Yaskawa INFORM job: R2_W27-A3(90,0)_MP_OK.JBI

/JOB
//NAME R2_W27-A3(90,0)_MP_OK
///FOLDERNAME MP_TEST
//POS
///NPOS 44,44,0,2,0,0
///TOOL 0
///POSTYPE PULSE
///PULSE
C00000=101600,-116692,-81613,16390,61564,19311
C00001=164215,-55536,-44539,-18349,62898,27662
C00002=160924,-13115,576,-12085,68568,20289
C00003=160935,-12305,2800,-12163,67637,20390
C00004=160940,-12317,2798,-12164,67633,20392
C00005=160946,-12330,2788,-12165,67634,20394
C00006=160940,-12317,2798,-12164,67633,20392
C00007=160931,-12288,2814,-12162,67637,20389
C00008=160930,-12287,2823,-12162,67632,20389
C00009=160931,-12288,2814,-12162,67637,20389
C00010=160981,-12434,2698,-978,54579,-1424
C00011=160979,-12429,2730,-978,54561,-1425
C00012=160976,-12421,2736,-977,54562,-1426
C00013=160979,-12429,2730,-978,54561,-1425
C00014=160981,-12434,2698,-978,54579,-1424
C00015=160997,-12478,2668,-985,54575,-1417
C00016=160994,-12473,2666,-984,54579,-1419
C00017=160987,-12460,2661,-981,54588,-1422
C00018=145436,-5822,-19148,1406,76142,21143
C00019=161005,-17259,-14065,-3869,52708,76882
C00020=161000,-11415,3879,-4366,44687,77223
C00021=161004,-11424,3871,-4369,44687,77225
C00022=165127,-14952,4261,-15285,39692,81657
C00023=161056,-12333,1868,-4344,45453,77213
C00024=160458,-11230,5111,-4075,43997,76999
C00025=163098,-8602,9142,-13757,39586,80598
C00026=161003,-11423,3872,-4369,44687,77225
C00027=160999,-11413,3880,-4366,44687,77223
C00028=161005,-17410,-14659,-3854,52995,76871
C00029=116418,-11777,-44439,19300,59296,60154
C00030=170009,-32177,-45595,-27188,83944,54223
C00031=188971,-7216,-15050,-32227,103013,52664
C00032=187803,-7888,-16310,-32403,102934,52210
C00033=188364,-6082,-14100,-32286,102781,52484
C00034=188636,-9365,-17003,-32274,102969,52540
C00035=189413,-7325,-10428,-33924,100512,54745
C00036=189914,-7682,-12670,-35106,101599,55206
C00037=190540,-7572,-11965,-36074,101422,56128
C00038=193143,-7278,-8936,-40285,100522,60148
C00039=196044,-7471,-5630,-45187,99267,64707
C00040=192289,-11545,-19761,-34441,104887,54555
C00041=160924,-13115,576,-12085,68568,20289
C00042=164215,-55536,-44539,-18349,62898,27662
C00043=101600,-116692,-81613,16390,61564,19311
BC00000=282797,179500,1075171
BC00001=315243,149725,1075174
BC00002=326313,139566,1075175
BC00003=327306,134779,1064198
BC00004=327703,132864,1055897
BC00005=327690,132857,1047832
BC00006=327703,132864,1055897
BC00007=317158,132350,1053533
BC00008=317644,130094,1053548
BC00009=317158,132350,1053533
BC00010=354979,141253,1041870
BC00011=356652,133484,1041925
BC00012=354313,133016,1041973
BC00013=356652,133484,1041925
BC00014=354979,141253,1041870
BC00015=363025,141681,1030105
BC00016=364240,143651,1037263
BC00017=367279,148578,1055156
BC00018=320233,175848,913334
BC00019=353844,149726,1075175
BC00020=353886,149731,1052313
BC00021=353827,147577,1026510
BC00022=353804,146715,1016186
BC00023=353804,146715,1016188
BC00024=353804,146715,1016188
BC00025=353804,146715,1016186
BC00026=353799,139703,1029577
BC00027=353858,141857,1055381
BC00028=353816,141852,1075175
BC00029=253941,214275,713494
BC00030=305300,128666,812515
BC00031=329706,95698,858127
BC00032=329696,96061,851804
BC00033=329696,96061,851804
BC00034=329696,96061,851804
BC00035=329682,96606,842319
BC00036=329681,96639,841736
BC00037=329663,97291,830381
BC00038=329660,97348,828220
BC00039=329656,97223,825887
BC00040=329682,96606,842319
BC00041=326313,139566,1075175
BC00042=315243,149725,1075174
BC00043=282797,179500,1075171
///POSTYPE BASE
///RECTAN
///RCONF 0,0,0,0,1,0,0,0,0,0,0,0,0,0,0,0,0,0,0,0,0,0,0,0
P00006=2.006,1.622,-0.565,0.0000,0.0000,0.0000
///RCONF 0,0,0,0,0,0,0,0,0,0,0,0,0,0,0,0,0,0,0,0,0,0,0,0
P00014=4.542,-3.738,3.339,0.0000,0.0000,0.0000
//INST
///DATE 2023/11/16 10:45
///ATTR SC,RW
///GROUP1 RB1,BS1
NOP
'r2_W27-A3(90,0)
'
'Path S839
SFTOF
MOVJ C00000 BC00000 VJ=20.00
MOVJ C00001 BC00001 VJ=20.00
MOVL C00002 BC00002 V=100.0
MOVL C00003 BC00003 V=100.0
MOVL C00004 BC00004 V=60.0
REFP 3 C00005 BC00005
CALL JOB:SEARCH-R1
SET P014 P006
SFTON P014
MOVL C00006 BC00006 V=60.0
MOVL C00007 BC00007 V=60.0
REFP 3 C00008 BC00008
CALL JOB:SEARCH-R1
SET P014 P006
SFTON P014
MOVL C00009 BC00009 V=60.0
MOVL C00010 BC00010 V=100.0
MOVL C00011 BC00011 V=60.0
REFP 3 C00012 BC00012
CALL JOB:SEARCH-R1
SET P014 P006
SFTON P014
MOVL C00013 BC00013 V=60.0
MOVL C00014 BC00014 V=100.0
MOVL C00015 BC00015 V=100.0
MOVL C00016 BC00016 V=100.0
MOVL C00017 BC00017 V=100.0
'Path VIA886
SFTOF
MOVJ C00018 BC00018 VJ=20.00
'Path W840
SFTOF
SFTON P014
'ZA DUZA SZCZELINA
'ZA DUZA SZCZELINA
'ZA DUZA SZCZELINA
MOVJ C00019 BC00019 VJ=20.00
MOVJ C00020 BC00020 VJ=20.00
MOVL C00021 BC00021 V=100.0
MOVL C00022 BC00022 V=100.0 PL=0
REFP 1 C00023 BC00023
REFP 2 C00024 BC00024
MACRO1 MJ#(0) ARGF7
COMM ARCON
MOVL C00025 BC00025 V=11.2
COMM ARCOF
MOVL C00026 BC00026 V=100.0
MOVL C00027 BC00027 V=100.0
MOVL C00028 BC00028 V=100.0
SFTOF
'Path VIA888
SFTOF
MOVJ C00029 BC00029 VJ=20.00
'Path VIA887
SFTOF
MOVJ C00030 BC00030 VJ=20.00
'Path W841
SFTOF
SFTON P014
MOVL C00031 BC00031 V=100.0
MOVL C00032 BC00032 V=100.0 PL=0
REFP 1 C00033 BC00033
REFP 2 C00034 BC00034
MACRO1 MJ#(0) ARGF7
ARCON
MOVL C00035 BC00035 V=12.5
COMM MOVL C00036 BC00036 V=10.0
COMM MOVL C00037 BC00037 V=10.0
COMM MOVL C00038 BC00038 V=10.0
COMM MOVL C00039 BC00039 V=10.0
ARCOF
MOVL C00040 BC00040 V=100.0
MOVL C00041 BC00041 V=100.0
MOVJ C00042 BC00042 VJ=20.00
MOVJ C00043 BC00043 VJ=20.00
SFTOF
END
